FUNCTION_BLOCK GET_STRUCT_VALUE (* Service Interface Function Block Type *)
  (* Standard: 61499-2; Description: Copyright (c) 2018 fortiss GmbH This program and the accompanying materials are made available under the terms of the Eclipse Public License 2.0 which is available at https://www.eclipse.org/legal/epl-2.0/ SPDX-License-Identifier: EPL-2.0 *)
  (* Version 1.0, 2018-10-16, Jose Cabral *)
  (* Version 3.0, 2025-04-14, Patrick Aigner, changed package *)
  PACKAGE eclipse4diac::utils;
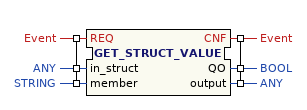
  EVENT_INPUT
    REQ WITH member, in_struct; (* Get Value out of structure *)
  END_EVENT
  EVENT_OUTPUT
    CNF WITH QO, output; (* REQ event finished *)
  END_EVENT
  VAR_INPUT
    in_struct : ANY; (* Structure to look into *)
    member : STRING; (* Member of the strucuture to retrieve. Inner members are access using the dot (.) operator *)
  END_VAR
  VAR_OUTPUT
    QO : BOOL; (* TRUE if no errors ocurred, FALSE otherwise *)
    output : ANY; (* Selected member if QO = TRUE, remains unchanged otherwise *)
  END_VAR
END_FUNCTION_BLOCK
